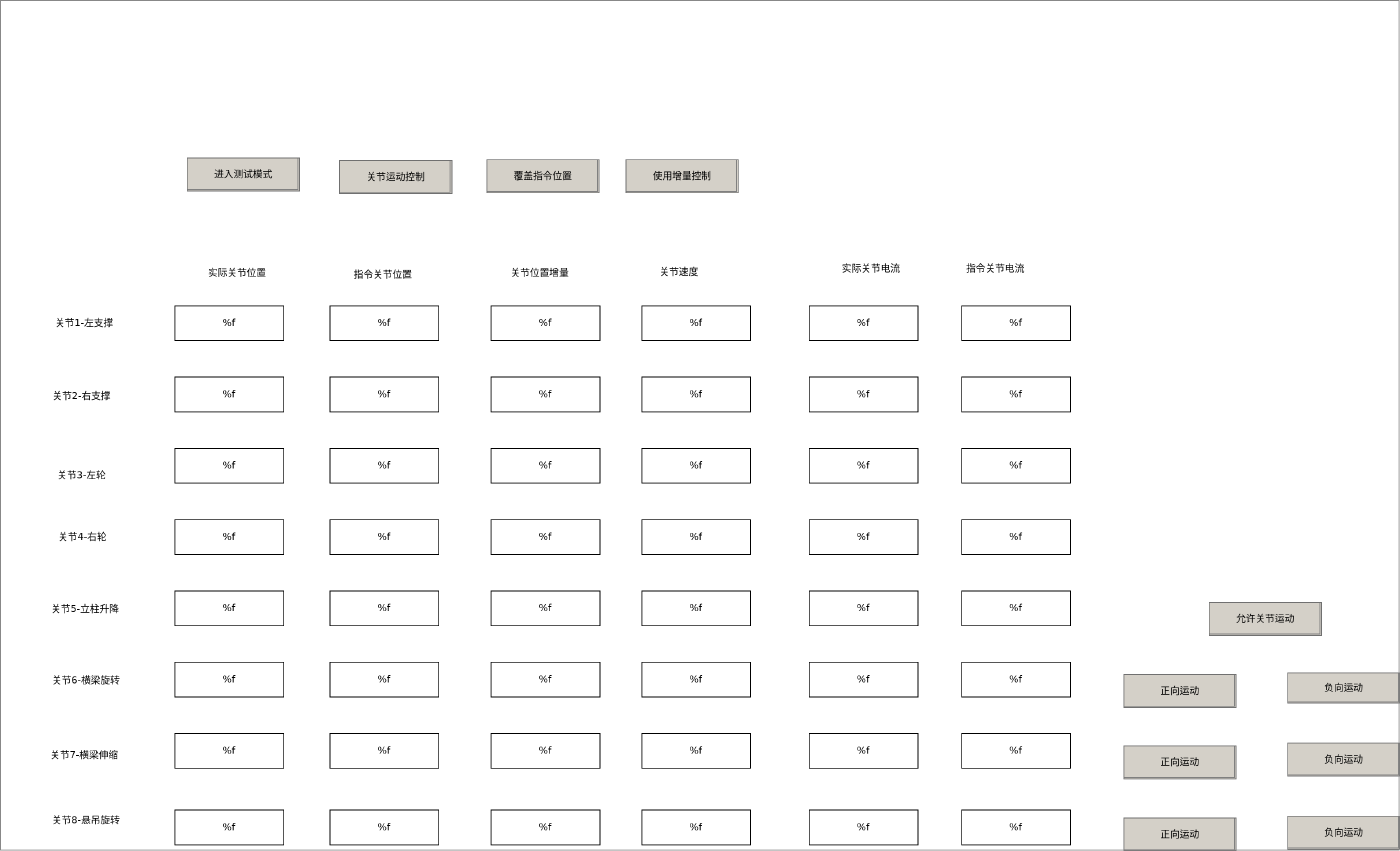
VISUALIZATION motion_car  // 1589x967
    Button (385,182 128x38), "关节运动控制", colour toggle: g_motionTest.m_uiArmModeCar[1]
        tap g_motionTest.m_uiArmModeCar[1]
    Button (212,179 128x38), "进入测试模式", colour toggle: g_motionTest.m_enterJntTestModeCar
        toggle g_motionTest.m_enterJntTestModeCar
    Label (362,298 145x28), "指令关节位置"
    Label (194,295 150x30), "实际关节位置"
    Label (540,296 145x28), "关节位置增量"
    Label (698,295 145x28), "关节速度"
    Label (916,291 145x28), "实际关节电流"
    Label (1057,291 145x28), "指令关节电流"
    Rectangle (198,590 124x40), "%f", text variable: g_motionTest.m_curJntPosCar[4]
    Label (23,353 145x28), "关节1-左支撑"
    Label (20,436 145x28), "关节2-右支撑"
    Label (20,526 145x28), "关节3-左轮"
    Label (21,596 145x28), "关节4-右轮"
    Label (24,678 145x28), "关节5-立柱升降"
    Label (25,759 145x28), "关节6-横梁旋转"
    Rectangle (198,671 124x40), "%f", text variable: g_motionTest.m_curJntPosCar[5]
    Rectangle (198,752 124x40), "%f", text variable: g_motionTest.m_curJntPosCar[6]
    Rectangle (198,347 124x40), "%f", text variable: g_motionTest.m_curJntPosCar[1]
    Rectangle (198,428 124x40), "%f", text variable: g_motionTest.m_curJntPosCar[2]
    Rectangle (198,509 124x40), "%f", text variable: g_motionTest.m_curJntPosCar[3]
    Rectangle (374,347 124x40), "%f", text variable: g_motionTest.m_targetJntPosCar[1]
        OnMouseClick: write the text variable via Default
    Rectangle (374,428 124x40), "%f", text variable: g_motionTest.m_targetJntPosCar[2]
        OnMouseClick: write the text variable via Default
    Rectangle (374,509 124x40), "%f", text variable: g_motionTest.m_targetJntPosCar[3]
        OnMouseClick: write the text variable via Default
    Rectangle (374,590 124x40), "%f", text variable: g_motionTest.m_targetJntPosCar[4]
        OnMouseClick: write the text variable via Default
    Rectangle (374,671 124x40), "%f", text variable: g_motionTest.m_targetJntPosCar[5]
        OnMouseClick: write the text variable via Default
    Rectangle (374,752 124x40), "%f", text variable: g_motionTest.m_targetJntPosCar[6]
        OnMouseClick: write the text variable via Default
    Rectangle (557,347 124x40), "%f", text variable: g_motionTest.m_targetJntPosIncCar[1]
        OnMouseClick: write the text variable via Default
    Rectangle (557,428 124x40), "%f", text variable: g_motionTest.m_targetJntPosIncCar[2]
        OnMouseClick: write the text variable via Default
    Rectangle (557,509 124x40), "%f", text variable: g_motionTest.m_targetJntPosIncCar[3]
        OnMouseClick: write the text variable via Default
    Rectangle (557,590 124x40), "%f", text variable: g_motionTest.m_targetJntPosIncCar[4]
        OnMouseClick: write the text variable via Default
    Rectangle (557,671 124x40), "%f", text variable: g_motionTest.m_targetJntPosIncCar[5]
        OnMouseClick: write the text variable via Default
    Rectangle (557,752 124x40), "%f", text variable: g_motionTest.m_targetJntPosIncCar[6]
        OnMouseClick: write the text variable via Default
    Rectangle (728,347 124x40), "%f", text variable: g_motionTest.m_targetJntVelCar[1]
        OnMouseClick: write the text variable via Default
    Rectangle (728,428 124x40), "%f", text variable: g_motionTest.m_targetJntVelCar[2]
        OnMouseClick: write the text variable via Default
    Rectangle (728,509 124x40), "%f", text variable: g_motionTest.m_targetJntVelCar[3]
        OnMouseClick: write the text variable via Default
    Rectangle (728,590 124x40), "%f", text variable: g_motionTest.m_targetJntVelCar[4]
        OnMouseClick: write the text variable via Default
    Rectangle (728,671 124x40), "%f", text variable: g_motionTest.m_targetJntVelCar[5]
        OnMouseClick: write the text variable via Default
    Rectangle (728,752 124x40), "%f", text variable: g_motionTest.m_targetJntVelCar[6]
        OnMouseClick: write the text variable via Default
    Rectangle (918,347 124x40), "%f", text variable: g_motionTest.m_curJntCurrentCar[1]
    Rectangle (918,428 124x40), "%f", text variable: g_motionTest.m_curJntCurrentCar[2]
    Rectangle (918,509 124x40), "%f", text variable: g_motionTest.m_curJntCurrentCar[3]
    Rectangle (918,590 124x40), "%f", text variable: g_motionTest.m_curJntCurrentCar[4]
    Rectangle (918,671 124x40), "%f", text variable: g_motionTest.m_curJntCurrentCar[5]
    Rectangle (918,752 124x40), "%f", text variable: g_motionTest.m_curJntCurrentCar[6]
    Rectangle (1091,347 124x40), "%f", text variable: g_motionTest.m_targetJntCurrentCar[1]
        OnMouseClick: write the text variable via Default
    Rectangle (1091,428 124x40), "%f", text variable: g_motionTest.m_targetJntCurrentCar[2]
        OnMouseClick: write the text variable via Default
    Rectangle (1091,509 124x40), "%f", text variable: g_motionTest.m_targetJntCurrentCar[3]
        OnMouseClick: write the text variable via Default
    Rectangle (1091,590 124x40), "%f", text variable: g_motionTest.m_targetJntCurrentCar[4]
        OnMouseClick: write the text variable via Default
    Rectangle (1091,671 124x40), "%f", text variable: g_motionTest.m_targetJntCurrentCar[5]
        OnMouseClick: write the text variable via Default
    Rectangle (1091,752 124x40), "%f", text variable: g_motionTest.m_targetJntCurrentCar[6]
        OnMouseClick: write the text variable via Default
    Button (710,181 128x38), "使用增量控制", colour toggle: g_motionTest.m_jntTestModeIncCar
        toggle g_motionTest.m_jntTestModeIncCar
    Button (1372,684 128x38), "允许关节运动", colour toggle: g_motionTest.m_uiArmModeCar[2]
        tap g_motionTest.m_uiArmModeCar[2]
    Rectangle (198,833 124x40), "%f", text variable: g_motionTest.m_curJntPosCar[7]
    Rectangle (198,920 124x40), "%f", text variable: g_motionTest.m_curJntPosCar[8]
    Rectangle (374,833 124x40), "%f", text variable: g_motionTest.m_targetJntPosCar[7]
        OnMouseClick: write the text variable via Default
    Rectangle (374,920 124x40), "%f", text variable: g_motionTest.m_targetJntPosCar[8]
        OnMouseClick: write the text variable via Default
    Rectangle (557,833 124x40), "%f", text variable: g_motionTest.m_targetJntPosIncCar[7]
        OnMouseClick: write the text variable via Default
    Rectangle (557,920 124x40), "%f", text variable: g_motionTest.m_targetJntPosIncCar[8]
        OnMouseClick: write the text variable via Default
    Rectangle (728,833 124x40), "%f", text variable: g_motionTest.m_targetJntVelCar[7]
        OnMouseClick: write the text variable via Default
    Rectangle (728,920 124x40), "%f", text variable: g_motionTest.m_targetJntVelCar[8]
        OnMouseClick: write the text variable via Default
    Rectangle (918,833 124x40), "%f", text variable: g_motionTest.m_curJntCurrentCar[7]
    Rectangle (918,920 124x40), "%f", text variable: g_motionTest.m_curJntCurrentCar[8]
    Rectangle (1091,833 124x40), "%f", text variable: g_motionTest.m_targetJntCurrentCar[7]
        OnMouseClick: write the text variable via Default
    Rectangle (1091,920 124x40), "%f", text variable: g_motionTest.m_targetJntCurrentCar[8]
        OnMouseClick: write the text variable via Default
    Label (23,844 145x28), "关节7-横梁伸缩"
    Label (25,918 145x28), "关节8-悬吊旋转"
    Button (1275,766 128x38), "正向运动", colour toggle: g_motionTest.m_caliMotPositive[6]
        toggle g_motionTest.m_caliMotPositive[6]
    Button (1461,764 128x35), "负向运动", colour toggle: g_motionTest.m_caliMotNegative[6]
        toggle g_motionTest.m_caliMotNegative[6]
    Button (1275,847 128x38), "正向运动", colour toggle: g_motionTest.m_caliMotPositive[7]
        toggle g_motionTest.m_caliMotPositive[7]
    Button (1461,844 128x38), "负向运动", colour toggle: g_motionTest.m_caliMotNegative[7]
        toggle g_motionTest.m_caliMotNegative[7]
    Button (1275,929 128x38), "正向运动", colour toggle: g_motionTest.m_caliMotPositive[8]
        toggle g_motionTest.m_caliMotPositive[8]
    Button (1461,927 128x38), "负向运动", colour toggle: g_motionTest.m_caliMotNegative[8]
        toggle g_motionTest.m_caliMotNegative[8]
    Button (552,181 128x38), "覆盖指令位置", colour toggle: g_motionTest.m_coverCmdPosCar
        tap g_motionTest.m_coverCmdPosCar
END_VISUALIZATION

(* stored: Version 1.1.0.1, ProductVersion 3.1.4024.11
   Visu motion_car: Id {bd855177-9b02-4a98-9d42-e0c6f6c07909} *)
